% RSLogix 500 project FINAL PROJECT_done.RSS, saved by version 8.40.00.08 %
PROJECT "UNTITLED"    % processor: MicroLogix 1000 %

PROGRAM FILES
  LAD 2 "MAIN_PROG"  31 rungs
  LAD 3 "USER_FAULT"  1 rungs
  LAD 4 "HSC_INT"  1 rungs
  LAD 5 "STI_INT"  1 rungs
  LAD 6, 7, 8, 9, 10, 11, 12, 13, 14, 15, 16: only END

DATA FILES
  O0 OUTPUT  1 elements
  I1 INPUT  2 elements
  S2 STATUS  33 elements
  B3 BINARY  32 elements
  T4 TIMER  40 elements
  C5 COUNTER  32 elements
  R6 CONTROL  16 elements
  N7 INTEGER  105 elements

LADDER 2 "MAIN_PROG"
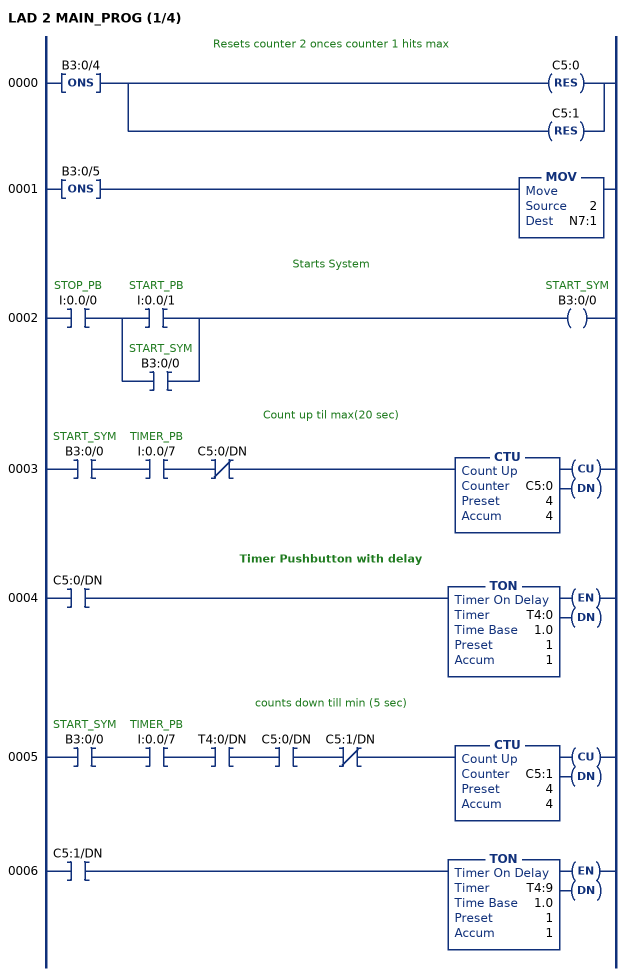
% Rung: 0 %
% Resets counter 2 onces counter 1 hits max %
SOR OSR B3:0/4 BST RES C5:0 NXB RES C5:1 BND EOR
% Rung: 1 %
SOR OSR B3:0/5 MOV 2 N7:1 EOR
% Rung: 2 %
% Starts System %
SOR XIC I:0.0/0 BST XIC I:0.0/1 NXB XIC B3:0/0 BND OTE B3:0/0 EOR
%   I:0.0/0  STOP_PB %
%   I:0.0/1  START_PB %
%   B3:0/0  START_SYM %
% Rung: 3 %
% Count up til max(20 sec) %
SOR XIC B3:0/0 XIC I:0.0/7 XIO C5:0/DN CTU C5:0 4 4 EOR
%   B3:0/0  START_SYM %
%   I:0.0/7  TIMER_PB %
% Rung: 4 %
% TITLE: Timer Pushbutton with delay %
SOR XIC C5:0/DN TON T4:0 1.0 1 1 EOR
% Rung: 5 %
% counts down till min (5 sec) %
SOR XIC B3:0/0 XIC I:0.0/7 XIC T4:0/DN XIC C5:0/DN XIO C5:1/DN CTU C5:1 4 4 EOR
%   B3:0/0  START_SYM %
%   I:0.0/7  TIMER_PB %
% Rung: 6 %
SOR XIC C5:1/DN TON T4:9 1.0 1 1 EOR

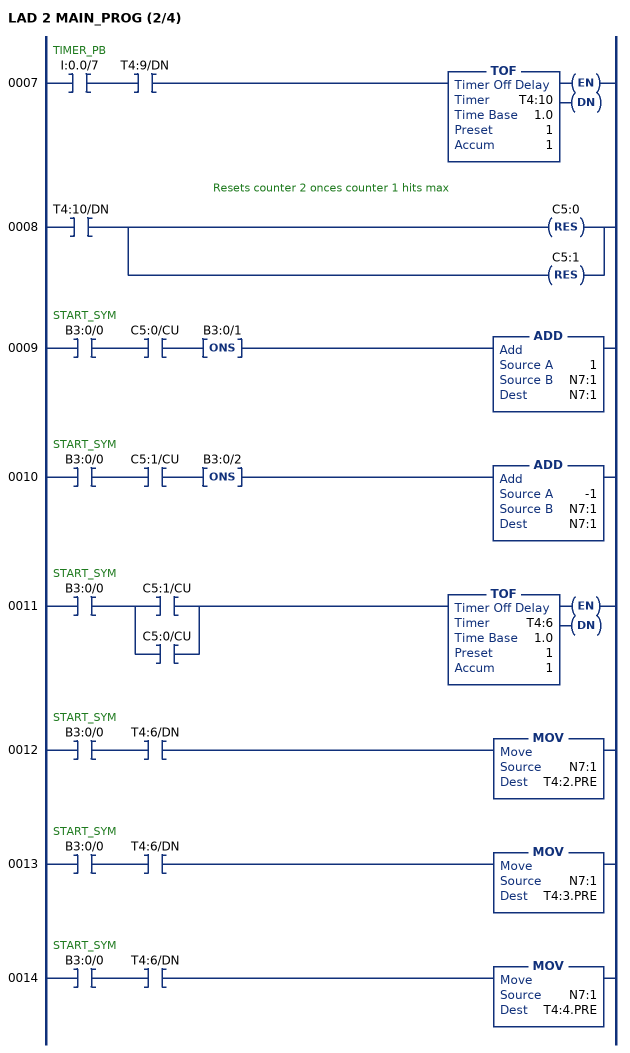
% Rung: 7 %
SOR XIC I:0.0/7 XIC T4:9/DN TOF T4:10 1.0 1 1 EOR
%   I:0.0/7  TIMER_PB %
% Rung: 8 %
% Resets counter 2 onces counter 1 hits max %
SOR XIC T4:10/DN BST RES C5:0 NXB RES C5:1 BND EOR
% Rung: 9 %
SOR XIC B3:0/0 XIC C5:0/CU OSR B3:0/1 ADD 1 N7:1 N7:1 EOR
%   B3:0/0  START_SYM %
% Rung: 10 %
SOR XIC B3:0/0 XIC C5:1/CU OSR B3:0/2 ADD -1 N7:1 N7:1 EOR
%   B3:0/0  START_SYM %
% Rung: 11 %
SOR XIC B3:0/0 BST XIC C5:1/CU NXB XIC C5:0/CU BND TOF T4:6 1.0 1 1 EOR
%   B3:0/0  START_SYM %
% Rung: 12 %
SOR XIC B3:0/0 XIC T4:6/DN MOV N7:1 T4:2.PRE EOR
%   B3:0/0  START_SYM %
% Rung: 13 %
SOR XIC B3:0/0 XIC T4:6/DN MOV N7:1 T4:3.PRE EOR
%   B3:0/0  START_SYM %
% Rung: 14 %
SOR XIC B3:0/0 XIC T4:6/DN MOV N7:1 T4:4.PRE EOR
%   B3:0/0  START_SYM %

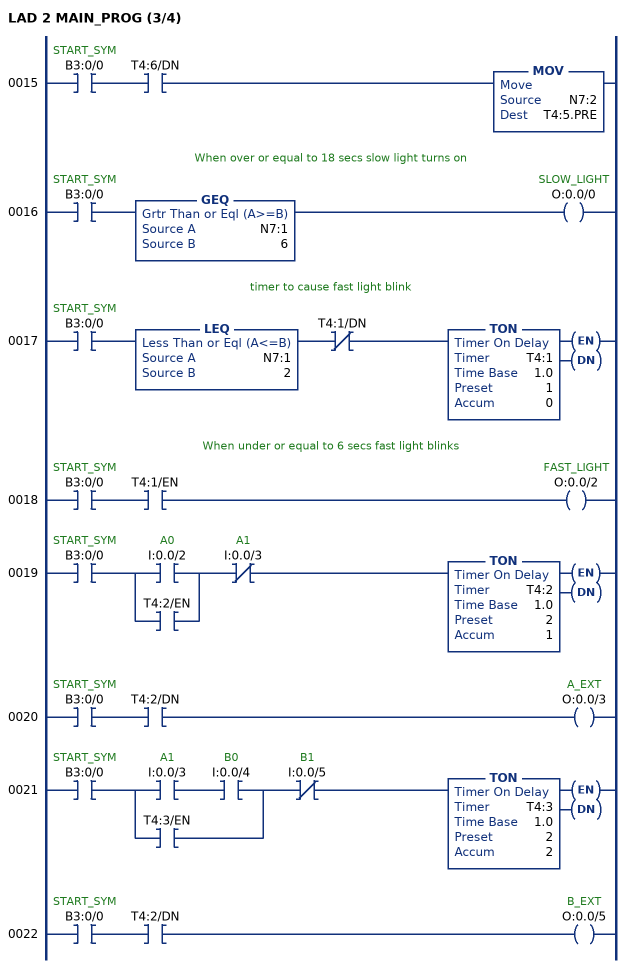
% Rung: 15 %
SOR XIC B3:0/0 XIC T4:6/DN MOV N7:2 T4:5.PRE EOR
%   B3:0/0  START_SYM %
% Rung: 16 %
% When over or equal to 18 secs slow light turns on %
SOR XIC B3:0/0 GEQ N7:1 6 OTE O:0.0/0 EOR
%   B3:0/0  START_SYM %
%   O:0.0/0  SLOW_LIGHT %
% Rung: 17 %
% timer to cause fast light blink %
SOR XIC B3:0/0 LEQ N7:1 2 XIO T4:1/DN TON T4:1 1.0 1 0 EOR
%   B3:0/0  START_SYM %
% Rung: 18 %
% When under or equal to 6 secs fast light blinks %
SOR XIC B3:0/0 XIC T4:1/EN OTE O:0.0/2 EOR
%   B3:0/0  START_SYM %
%   O:0.0/2  FAST_LIGHT %
% Rung: 19 %
SOR XIC B3:0/0 BST XIC I:0.0/2 NXB XIC T4:2/EN BND XIO I:0.0/3 TON T4:2 1.0 2 1 EOR
%   B3:0/0  START_SYM %
%   I:0.0/2  A0 %
%   I:0.0/3  A1 %
% Rung: 20 %
SOR XIC B3:0/0 XIC T4:2/DN OTE O:0.0/3 EOR
%   B3:0/0  START_SYM %
%   O:0.0/3  A_EXT %
% Rung: 21 %
SOR XIC B3:0/0 BST XIC I:0.0/3 XIC I:0.0/4 NXB XIC T4:3/EN BND XIO I:0.0/5 TON T4:3 1.0 2 2 EOR
%   B3:0/0  START_SYM %
%   I:0.0/3  A1 %
%   I:0.0/4  B0 %
%   I:0.0/5  B1 %
% Rung: 22 %
SOR XIC B3:0/0 XIC T4:2/DN OTE O:0.0/5 EOR
%   B3:0/0  START_SYM %
%   O:0.0/5  B_EXT %

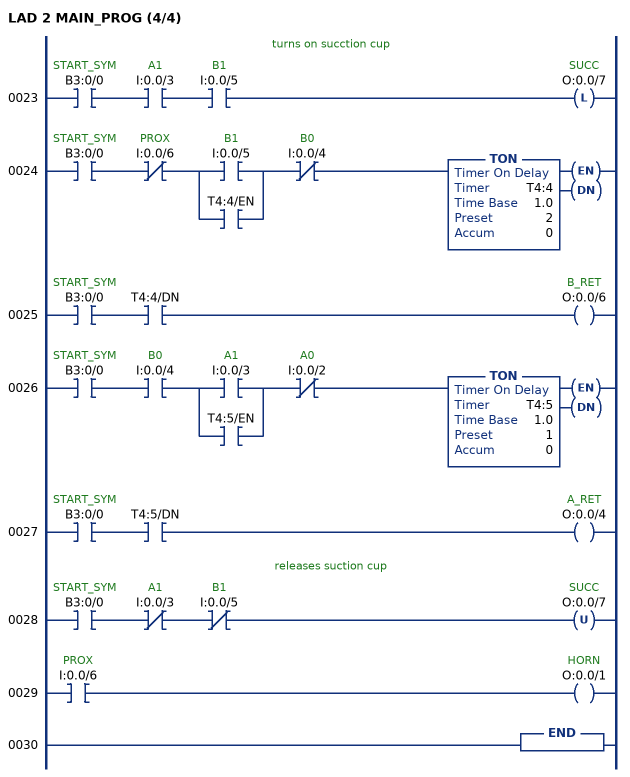
% Rung: 23 %
% turns on sucction cup %
SOR XIC B3:0/0 XIC I:0.0/3 XIC I:0.0/5 OTL O:0.0/7 EOR
%   B3:0/0  START_SYM %
%   I:0.0/3  A1 %
%   I:0.0/5  B1 %
%   O:0.0/7  SUCC %
% Rung: 24 %
SOR XIC B3:0/0 XIO I:0.0/6 BST XIC I:0.0/5 NXB XIC T4:4/EN BND XIO I:0.0/4 TON T4:4 1.0 2 0 EOR
%   B3:0/0  START_SYM %
%   I:0.0/6  PROX %
%   I:0.0/5  B1 %
%   I:0.0/4  B0 %
% Rung: 25 %
SOR XIC B3:0/0 XIC T4:4/DN OTE O:0.0/6 EOR
%   B3:0/0  START_SYM %
%   O:0.0/6  B_RET %
% Rung: 26 %
SOR XIC B3:0/0 XIC I:0.0/4 BST XIC I:0.0/3 NXB XIC T4:5/EN BND XIO I:0.0/2 TON T4:5 1.0 1 0 EOR
%   B3:0/0  START_SYM %
%   I:0.0/4  B0 %
%   I:0.0/3  A1 %
%   I:0.0/2  A0 %
% Rung: 27 %
SOR XIC B3:0/0 XIC T4:5/DN OTE O:0.0/4 EOR
%   B3:0/0  START_SYM %
%   O:0.0/4  A_RET %
% Rung: 28 %
% releases suction cup %
SOR XIC B3:0/0 XIO I:0.0/3 XIO I:0.0/5 OTU O:0.0/7 EOR
%   B3:0/0  START_SYM %
%   I:0.0/3  A1 %
%   I:0.0/5  B1 %
%   O:0.0/7  SUCC %
% Rung: 29 %
SOR XIC I:0.0/6 OTE O:0.0/1 EOR
%   I:0.0/6  PROX %
%   O:0.0/1  HORN %
% Rung: 30 %
SOR END EOR

OTHER DOCUMENTED ADDRESSES
  T0:0  T0

COMMENTS NOT ATTACHED TO A CURRENT RUNG
  B3:0/0: Starts System
  C5:0: Resets counter 1 onces counter 2 hits max

DATA TABLE (non-zero values as saved)
DATA B3
% B3:0 % 0X0031 0X0000 0X0000 0X0000 0X0000 0X0000 0X0000 0X0000 0X0000 0X0000
DATA T4
% .PRE .ACC %
% T4:0 % 1 1
% T4:1 % 1 0
% T4:2 % 2 1
% T4:3 % 2 2
% T4:4 % 2 0
% T4:5 % 1 0
% T4:6 % 1 1
% T4:8 % 1 0
% T4:9 % 1 1
% T4:10 % 1 1
DATA C5
% .PRE .ACC %
% C5:0 % 4 4
% C5:1 % 4 4
DATA N7
% N7:0 % 0 2 1 0 0 0 0 0 0 0
